REGION Network 163: ACKNOWLEDGE M573-
   RUNG wire#powerrail
      Contact( "M_ZERO" )
      Coil( "DB371_M_UNIT_SPARE".M_CODES_SPARE.Ack_M573 )
   END_RUNG
   // the same network as SCL:
   "DB371_M_UNIT_SPARE".M_CODES_SPARE.Ack_M573 := "M_ZERO";
END_REGION

REGION Network 164: M573-
   RUNG wire#powerrail
      Contact( "DB339_EXTENDED_M_SPARE".M_code[573] )
      wire#w1
      I_Contact( "DB371_M_UNIT_SPARE".M_CODES_SPARE.Ack_M573 )
      I_Contact( "DB2120_MPP_ITC_IPC".RESET_FAULTS )
      I_Contact( "DB371_M_UNIT_SPARE".M_CODES_SPARE.M_RESET_PULSE )
      Coil( "DB371_M_UNIT_SPARE".M_CODES_SPARE.M573 )
   END_RUNG
   RUNG wire#powerrail
      Contact( "DB371_M_UNIT_SPARE".M_CODES_SPARE.M573 )
   END_RUNG wire#w1
   // the same network as SCL:
   "DB371_M_UNIT_SPARE".M_CODES_SPARE.M573 := ("DB339_EXTENDED_M_SPARE".M_code[573] OR "DB371_M_UNIT_SPARE".M_CODES_SPARE.M573) AND NOT "DB371_M_UNIT_SPARE".M_CODES_SPARE.Ack_M573 AND NOT "DB2120_MPP_ITC_IPC".RESET_FAULTS AND NOT "DB371_M_UNIT_SPARE".M_CODES_SPARE.M_RESET_PULSE;
END_REGION

REGION Network 165: ACKNOWLEDGE M574- (READ-IN DISABLE)
   RUNG wire#powerrail
      Contact( "M_ZERO" )
      Coil( "DB371_M_UNIT_SPARE".M_CODES_SPARE.Ack_M574 )
   END_RUNG
   // the same network as SCL:
   "DB371_M_UNIT_SPARE".M_CODES_SPARE.Ack_M574 := "M_ZERO";
END_REGION

REGION Network 166: M574- (READ-IN DISABLE)
   RUNG wire#powerrail
      Contact( "DB339_EXTENDED_M_SPARE".M_code[574] )
      wire#w1
      I_Contact( "DB371_M_UNIT_SPARE".M_CODES_SPARE.Ack_M574 )
      I_Contact( "DB2120_MPP_ITC_IPC".RESET_FAULTS )
      I_Contact( "DB371_M_UNIT_SPARE".M_CODES_SPARE.M_RESET_PULSE )
      Coil( "DB371_M_UNIT_SPARE".M_CODES_SPARE.M574 )
   END_RUNG
   RUNG wire#powerrail
      Contact( "DB371_M_UNIT_SPARE".M_CODES_SPARE.M574 )
   END_RUNG wire#w1
   // the same network as SCL:
   "DB371_M_UNIT_SPARE".M_CODES_SPARE.M574 := ("DB339_EXTENDED_M_SPARE".M_code[574] OR "DB371_M_UNIT_SPARE".M_CODES_SPARE.M574) AND NOT "DB371_M_UNIT_SPARE".M_CODES_SPARE.Ack_M574 AND NOT "DB2120_MPP_ITC_IPC".RESET_FAULTS AND NOT "DB371_M_UNIT_SPARE".M_CODES_SPARE.M_RESET_PULSE;
END_REGION

REGION Network 167: ACKNOWLEDGE M575-(READ-IN DISABLE) / ACKNOWLEDGE M23-SWITCH ON SPINDLE FRAME BLOWING
   RUNG wire#powerrail
      Contact( "M_ZERO" )
      Coil( "DB371_M_UNIT_SPARE".M_CODES_SPARE.Ack_M575 )
   END_RUNG
   // the same network as SCL:
   "DB371_M_UNIT_SPARE".M_CODES_SPARE.Ack_M575 := "M_ZERO";
END_REGION

REGION Network 168: M575-(READ-IN DISABLE) / M23-SWITCH ON SPINDLE FRAME BLOWING
   RUNG wire#powerrail
      Contact( "DB339_EXTENDED_M_SPARE".M_code[575] )
      wire#w1
      I_Contact( "DB371_M_UNIT_SPARE".M_CODES_SPARE.Ack_M575 )
      I_Contact( "DB2120_MPP_ITC_IPC".RESET_FAULTS )
      I_Contact( "DB371_M_UNIT_SPARE".M_CODES_SPARE.M_RESET_PULSE )
      Coil( "DB371_M_UNIT_SPARE".M_CODES_SPARE.M575 )
   END_RUNG
   RUNG wire#powerrail
      Contact( "DB371_M_UNIT_SPARE".M_CODES_SPARE.M575 )
   END_RUNG wire#w1
   // the same network as SCL:
   "DB371_M_UNIT_SPARE".M_CODES_SPARE.M575 := ("DB339_EXTENDED_M_SPARE".M_code[575] OR "DB371_M_UNIT_SPARE".M_CODES_SPARE.M575) AND NOT "DB371_M_UNIT_SPARE".M_CODES_SPARE.Ack_M575 AND NOT "DB2120_MPP_ITC_IPC".RESET_FAULTS AND NOT "DB371_M_UNIT_SPARE".M_CODES_SPARE.M_RESET_PULSE;
END_REGION

REGION Network 169: ACKNOWLEDGE M588- (READ-IN DISABLE) / ACKNOWLEDGE M23-SWITCH ON SPINDLE FRAME BLOWING
   RUNG wire#powerrail
      Contact( "M_ZERO" )
      Coil( "DB371_M_UNIT_SPARE".M_CODES_SPARE.Ack_M588 )
   END_RUNG
   // the same network as SCL:
   "DB371_M_UNIT_SPARE".M_CODES_SPARE.Ack_M588 := "M_ZERO";
END_REGION

REGION Network 170: M588-(READ-IN DISABLE) / M23-SWITCH ON SPINDLE FRAME BLOWING
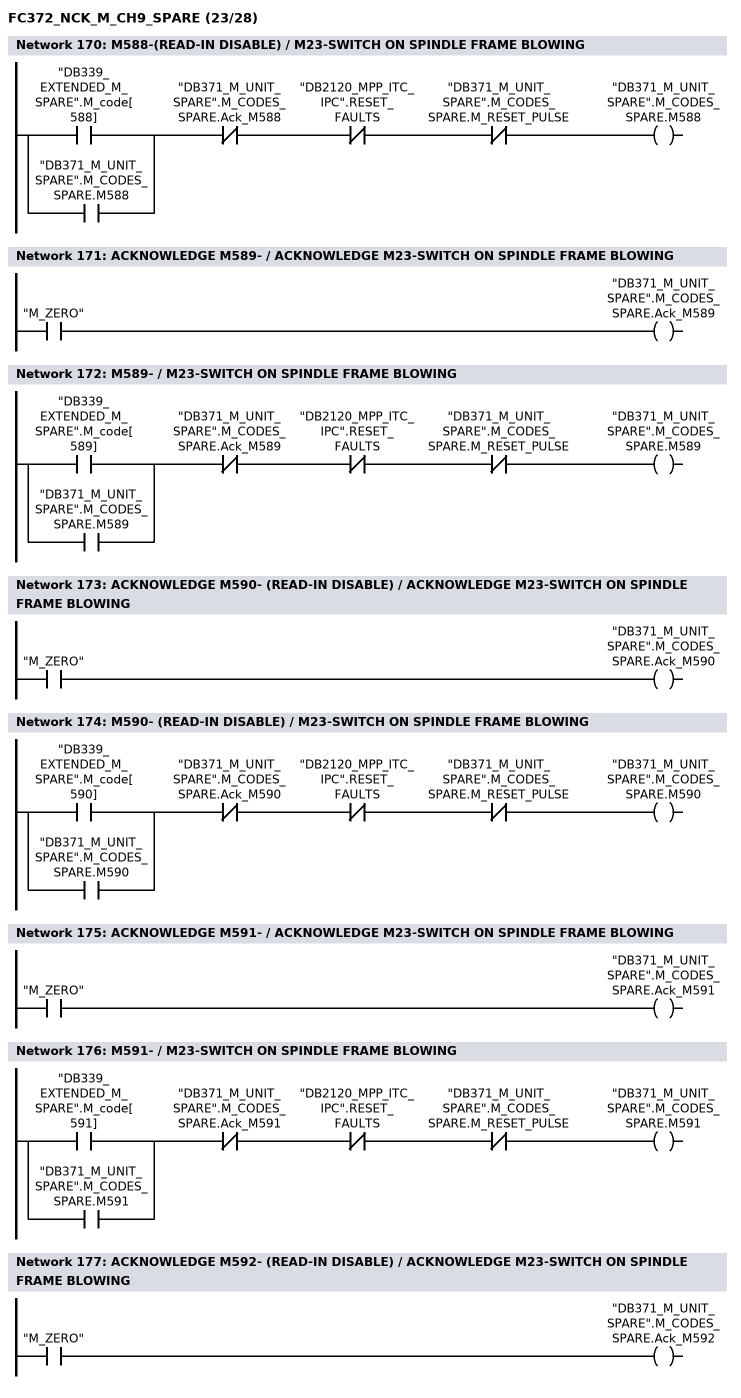
   RUNG wire#powerrail
      Contact( "DB339_EXTENDED_M_SPARE".M_code[588] )
      wire#w1
      I_Contact( "DB371_M_UNIT_SPARE".M_CODES_SPARE.Ack_M588 )
      I_Contact( "DB2120_MPP_ITC_IPC".RESET_FAULTS )
      I_Contact( "DB371_M_UNIT_SPARE".M_CODES_SPARE.M_RESET_PULSE )
      Coil( "DB371_M_UNIT_SPARE".M_CODES_SPARE.M588 )
   END_RUNG
   RUNG wire#powerrail
      Contact( "DB371_M_UNIT_SPARE".M_CODES_SPARE.M588 )
   END_RUNG wire#w1
   // the same network as SCL:
   "DB371_M_UNIT_SPARE".M_CODES_SPARE.M588 := ("DB339_EXTENDED_M_SPARE".M_code[588] OR "DB371_M_UNIT_SPARE".M_CODES_SPARE.M588) AND NOT "DB371_M_UNIT_SPARE".M_CODES_SPARE.Ack_M588 AND NOT "DB2120_MPP_ITC_IPC".RESET_FAULTS AND NOT "DB371_M_UNIT_SPARE".M_CODES_SPARE.M_RESET_PULSE;
END_REGION

REGION Network 171: ACKNOWLEDGE M589- / ACKNOWLEDGE M23-SWITCH ON SPINDLE FRAME BLOWING
   RUNG wire#powerrail
      Contact( "M_ZERO" )
      Coil( "DB371_M_UNIT_SPARE".M_CODES_SPARE.Ack_M589 )
   END_RUNG
   // the same network as SCL:
   "DB371_M_UNIT_SPARE".M_CODES_SPARE.Ack_M589 := "M_ZERO";
END_REGION

REGION Network 172: M589- / M23-SWITCH ON SPINDLE FRAME BLOWING
   RUNG wire#powerrail
      Contact( "DB339_EXTENDED_M_SPARE".M_code[589] )
      wire#w1
      I_Contact( "DB371_M_UNIT_SPARE".M_CODES_SPARE.Ack_M589 )
      I_Contact( "DB2120_MPP_ITC_IPC".RESET_FAULTS )
      I_Contact( "DB371_M_UNIT_SPARE".M_CODES_SPARE.M_RESET_PULSE )
      Coil( "DB371_M_UNIT_SPARE".M_CODES_SPARE.M589 )
   END_RUNG
   RUNG wire#powerrail
      Contact( "DB371_M_UNIT_SPARE".M_CODES_SPARE.M589 )
   END_RUNG wire#w1
   // the same network as SCL:
   "DB371_M_UNIT_SPARE".M_CODES_SPARE.M589 := ("DB339_EXTENDED_M_SPARE".M_code[589] OR "DB371_M_UNIT_SPARE".M_CODES_SPARE.M589) AND NOT "DB371_M_UNIT_SPARE".M_CODES_SPARE.Ack_M589 AND NOT "DB2120_MPP_ITC_IPC".RESET_FAULTS AND NOT "DB371_M_UNIT_SPARE".M_CODES_SPARE.M_RESET_PULSE;
END_REGION

REGION Network 173: ACKNOWLEDGE M590- (READ-IN DISABLE) / ACKNOWLEDGE M23-SWITCH ON SPINDLE FRAME BLOWING
   RUNG wire#powerrail
      Contact( "M_ZERO" )
      Coil( "DB371_M_UNIT_SPARE".M_CODES_SPARE.Ack_M590 )
   END_RUNG
   // the same network as SCL:
   "DB371_M_UNIT_SPARE".M_CODES_SPARE.Ack_M590 := "M_ZERO";
END_REGION

REGION Network 174: M590- (READ-IN DISABLE) / M23-SWITCH ON SPINDLE FRAME BLOWING
   RUNG wire#powerrail
      Contact( "DB339_EXTENDED_M_SPARE".M_code[590] )
      wire#w1
      I_Contact( "DB371_M_UNIT_SPARE".M_CODES_SPARE.Ack_M590 )
      I_Contact( "DB2120_MPP_ITC_IPC".RESET_FAULTS )
      I_Contact( "DB371_M_UNIT_SPARE".M_CODES_SPARE.M_RESET_PULSE )
      Coil( "DB371_M_UNIT_SPARE".M_CODES_SPARE.M590 )
   END_RUNG
   RUNG wire#powerrail
      Contact( "DB371_M_UNIT_SPARE".M_CODES_SPARE.M590 )
   END_RUNG wire#w1
   // the same network as SCL:
   "DB371_M_UNIT_SPARE".M_CODES_SPARE.M590 := ("DB339_EXTENDED_M_SPARE".M_code[590] OR "DB371_M_UNIT_SPARE".M_CODES_SPARE.M590) AND NOT "DB371_M_UNIT_SPARE".M_CODES_SPARE.Ack_M590 AND NOT "DB2120_MPP_ITC_IPC".RESET_FAULTS AND NOT "DB371_M_UNIT_SPARE".M_CODES_SPARE.M_RESET_PULSE;
END_REGION

REGION Network 175: ACKNOWLEDGE M591- / ACKNOWLEDGE M23-SWITCH ON SPINDLE FRAME BLOWING
   RUNG wire#powerrail
      Contact( "M_ZERO" )
      Coil( "DB371_M_UNIT_SPARE".M_CODES_SPARE.Ack_M591 )
   END_RUNG
   // the same network as SCL:
   "DB371_M_UNIT_SPARE".M_CODES_SPARE.Ack_M591 := "M_ZERO";
END_REGION

REGION Network 176: M591- / M23-SWITCH ON SPINDLE FRAME BLOWING
   RUNG wire#powerrail
      Contact( "DB339_EXTENDED_M_SPARE".M_code[591] )
      wire#w1
      I_Contact( "DB371_M_UNIT_SPARE".M_CODES_SPARE.Ack_M591 )
      I_Contact( "DB2120_MPP_ITC_IPC".RESET_FAULTS )
      I_Contact( "DB371_M_UNIT_SPARE".M_CODES_SPARE.M_RESET_PULSE )
      Coil( "DB371_M_UNIT_SPARE".M_CODES_SPARE.M591 )
   END_RUNG
   RUNG wire#powerrail
      Contact( "DB371_M_UNIT_SPARE".M_CODES_SPARE.M591 )
   END_RUNG wire#w1
   // the same network as SCL:
   "DB371_M_UNIT_SPARE".M_CODES_SPARE.M591 := ("DB339_EXTENDED_M_SPARE".M_code[591] OR "DB371_M_UNIT_SPARE".M_CODES_SPARE.M591) AND NOT "DB371_M_UNIT_SPARE".M_CODES_SPARE.Ack_M591 AND NOT "DB2120_MPP_ITC_IPC".RESET_FAULTS AND NOT "DB371_M_UNIT_SPARE".M_CODES_SPARE.M_RESET_PULSE;
END_REGION

REGION Network 177: ACKNOWLEDGE M592- (READ-IN DISABLE) / ACKNOWLEDGE M23-SWITCH ON SPINDLE FRAME BLOWING
   RUNG wire#powerrail
      Contact( "M_ZERO" )
      Coil( "DB371_M_UNIT_SPARE".M_CODES_SPARE.Ack_M592 )
   END_RUNG
   // the same network as SCL:
   "DB371_M_UNIT_SPARE".M_CODES_SPARE.Ack_M592 := "M_ZERO";
END_REGION

REGION Network 178: M592- (READ-IN DISABLE) / M23-SWITCH ON SPINDLE FRAME BLOWING
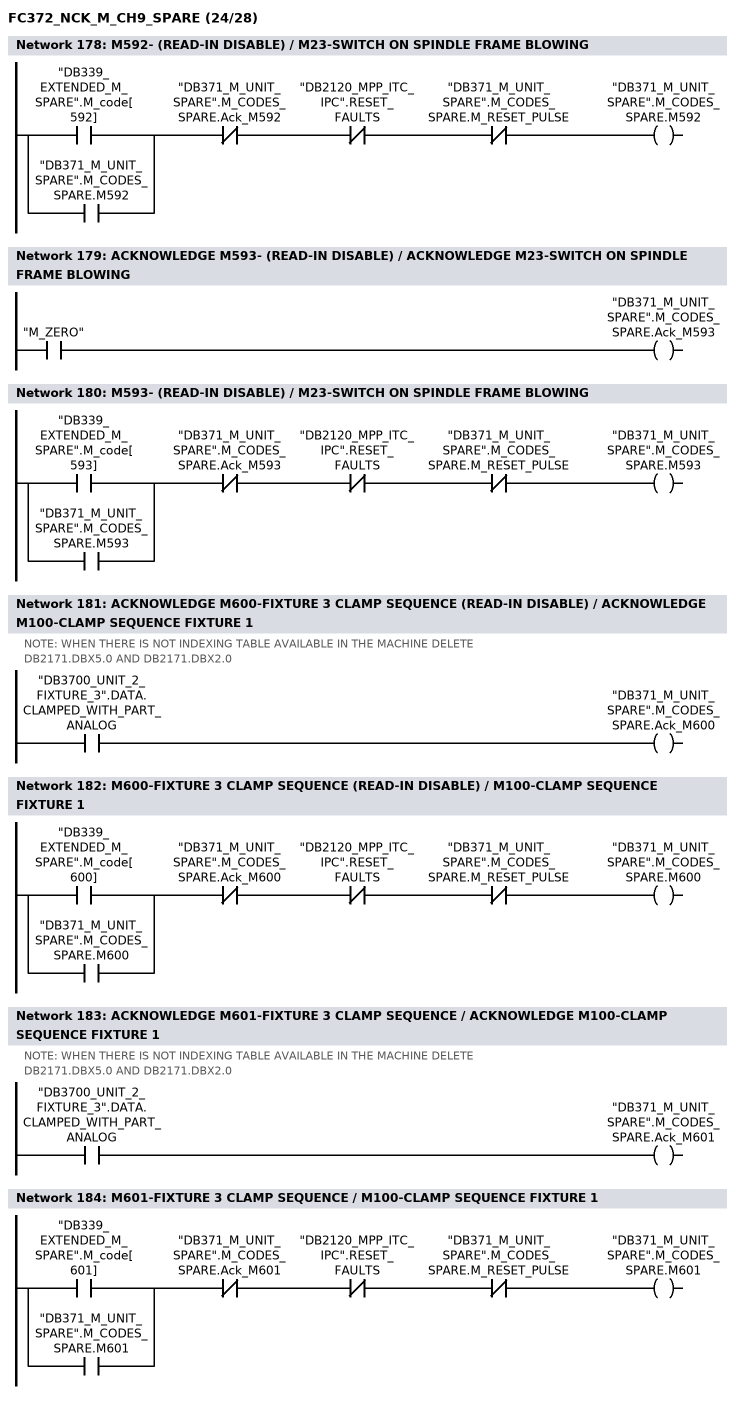
   RUNG wire#powerrail
      Contact( "DB339_EXTENDED_M_SPARE".M_code[592] )
      wire#w1
      I_Contact( "DB371_M_UNIT_SPARE".M_CODES_SPARE.Ack_M592 )
      I_Contact( "DB2120_MPP_ITC_IPC".RESET_FAULTS )
      I_Contact( "DB371_M_UNIT_SPARE".M_CODES_SPARE.M_RESET_PULSE )
      Coil( "DB371_M_UNIT_SPARE".M_CODES_SPARE.M592 )
   END_RUNG
   RUNG wire#powerrail
      Contact( "DB371_M_UNIT_SPARE".M_CODES_SPARE.M592 )
   END_RUNG wire#w1
   // the same network as SCL:
   "DB371_M_UNIT_SPARE".M_CODES_SPARE.M592 := ("DB339_EXTENDED_M_SPARE".M_code[592] OR "DB371_M_UNIT_SPARE".M_CODES_SPARE.M592) AND NOT "DB371_M_UNIT_SPARE".M_CODES_SPARE.Ack_M592 AND NOT "DB2120_MPP_ITC_IPC".RESET_FAULTS AND NOT "DB371_M_UNIT_SPARE".M_CODES_SPARE.M_RESET_PULSE;
END_REGION

REGION Network 179: ACKNOWLEDGE M593- (READ-IN DISABLE) / ACKNOWLEDGE M23-SWITCH ON SPINDLE FRAME BLOWING
   RUNG wire#powerrail
      Contact( "M_ZERO" )
      Coil( "DB371_M_UNIT_SPARE".M_CODES_SPARE.Ack_M593 )
   END_RUNG
   // the same network as SCL:
   "DB371_M_UNIT_SPARE".M_CODES_SPARE.Ack_M593 := "M_ZERO";
END_REGION

REGION Network 180: M593- (READ-IN DISABLE) / M23-SWITCH ON SPINDLE FRAME BLOWING
   RUNG wire#powerrail
      Contact( "DB339_EXTENDED_M_SPARE".M_code[593] )
      wire#w1
      I_Contact( "DB371_M_UNIT_SPARE".M_CODES_SPARE.Ack_M593 )
      I_Contact( "DB2120_MPP_ITC_IPC".RESET_FAULTS )
      I_Contact( "DB371_M_UNIT_SPARE".M_CODES_SPARE.M_RESET_PULSE )
      Coil( "DB371_M_UNIT_SPARE".M_CODES_SPARE.M593 )
   END_RUNG
   RUNG wire#powerrail
      Contact( "DB371_M_UNIT_SPARE".M_CODES_SPARE.M593 )
   END_RUNG wire#w1
   // the same network as SCL:
   "DB371_M_UNIT_SPARE".M_CODES_SPARE.M593 := ("DB339_EXTENDED_M_SPARE".M_code[593] OR "DB371_M_UNIT_SPARE".M_CODES_SPARE.M593) AND NOT "DB371_M_UNIT_SPARE".M_CODES_SPARE.Ack_M593 AND NOT "DB2120_MPP_ITC_IPC".RESET_FAULTS AND NOT "DB371_M_UNIT_SPARE".M_CODES_SPARE.M_RESET_PULSE;
END_REGION

REGION Network 181: ACKNOWLEDGE M600-FIXTURE 3 CLAMP SEQUENCE (READ-IN DISABLE) / ACKNOWLEDGE M100-CLAMP SEQUENCE FIXTURE 1
   // NOTE: WHEN THERE IS NOT INDEXING TABLE AVAILABLE IN THE MACHINE DELETE 
   // DB2171.DBX5.0 AND DB2171.DBX2.0
   RUNG wire#powerrail
      Contact( "DB3700_UNIT_2_FIXTURE_3".DATA.CLAMPED_WITH_PART_ANALOG )
      Coil( "DB371_M_UNIT_SPARE".M_CODES_SPARE.Ack_M600 )
   END_RUNG
   // the same network as SCL:
   "DB371_M_UNIT_SPARE".M_CODES_SPARE.Ack_M600 := "DB3700_UNIT_2_FIXTURE_3".DATA.CLAMPED_WITH_PART_ANALOG;
END_REGION

REGION Network 182: M600-FIXTURE 3 CLAMP SEQUENCE (READ-IN DISABLE) / M100-CLAMP SEQUENCE FIXTURE 1
   RUNG wire#powerrail
      Contact( "DB339_EXTENDED_M_SPARE".M_code[600] )
      wire#w1
      I_Contact( "DB371_M_UNIT_SPARE".M_CODES_SPARE.Ack_M600 )
      I_Contact( "DB2120_MPP_ITC_IPC".RESET_FAULTS )
      I_Contact( "DB371_M_UNIT_SPARE".M_CODES_SPARE.M_RESET_PULSE )
      Coil( "DB371_M_UNIT_SPARE".M_CODES_SPARE.M600 )
   END_RUNG
   RUNG wire#powerrail
      Contact( "DB371_M_UNIT_SPARE".M_CODES_SPARE.M600 )
   END_RUNG wire#w1
   // the same network as SCL:
   "DB371_M_UNIT_SPARE".M_CODES_SPARE.M600 := ("DB339_EXTENDED_M_SPARE".M_code[600] OR "DB371_M_UNIT_SPARE".M_CODES_SPARE.M600) AND NOT "DB371_M_UNIT_SPARE".M_CODES_SPARE.Ack_M600 AND NOT "DB2120_MPP_ITC_IPC".RESET_FAULTS AND NOT "DB371_M_UNIT_SPARE".M_CODES_SPARE.M_RESET_PULSE;
END_REGION

REGION Network 183: ACKNOWLEDGE M601-FIXTURE 3 CLAMP SEQUENCE / ACKNOWLEDGE M100-CLAMP SEQUENCE FIXTURE 1
   // NOTE: WHEN THERE IS NOT INDEXING TABLE AVAILABLE IN THE MACHINE DELETE 
   // DB2171.DBX5.0 AND DB2171.DBX2.0
   RUNG wire#powerrail
      Contact( "DB3700_UNIT_2_FIXTURE_3".DATA.CLAMPED_WITH_PART_ANALOG )
      Coil( "DB371_M_UNIT_SPARE".M_CODES_SPARE.Ack_M601 )
   END_RUNG
   // the same network as SCL:
   "DB371_M_UNIT_SPARE".M_CODES_SPARE.Ack_M601 := "DB3700_UNIT_2_FIXTURE_3".DATA.CLAMPED_WITH_PART_ANALOG;
END_REGION

REGION Network 184: M601-FIXTURE 3 CLAMP SEQUENCE / M100-CLAMP SEQUENCE FIXTURE 1
   RUNG wire#powerrail
      Contact( "DB339_EXTENDED_M_SPARE".M_code[601] )
      wire#w1
      I_Contact( "DB371_M_UNIT_SPARE".M_CODES_SPARE.Ack_M601 )
      I_Contact( "DB2120_MPP_ITC_IPC".RESET_FAULTS )
      I_Contact( "DB371_M_UNIT_SPARE".M_CODES_SPARE.M_RESET_PULSE )
      Coil( "DB371_M_UNIT_SPARE".M_CODES_SPARE.M601 )
   END_RUNG
   RUNG wire#powerrail
      Contact( "DB371_M_UNIT_SPARE".M_CODES_SPARE.M601 )
   END_RUNG wire#w1
   // the same network as SCL:
   "DB371_M_UNIT_SPARE".M_CODES_SPARE.M601 := ("DB339_EXTENDED_M_SPARE".M_code[601] OR "DB371_M_UNIT_SPARE".M_CODES_SPARE.M601) AND NOT "DB371_M_UNIT_SPARE".M_CODES_SPARE.Ack_M601 AND NOT "DB2120_MPP_ITC_IPC".RESET_FAULTS AND NOT "DB371_M_UNIT_SPARE".M_CODES_SPARE.M_RESET_PULSE;
END_REGION

REGION Network 185: ACKNOWLEDGE M602-FIXTURE 3 UNCLAMP SEQUENCE (READ-IN DISABLE) / ACKNOWLEDGE M101-UNCLAMP SEQUENCE FIXTURE 1
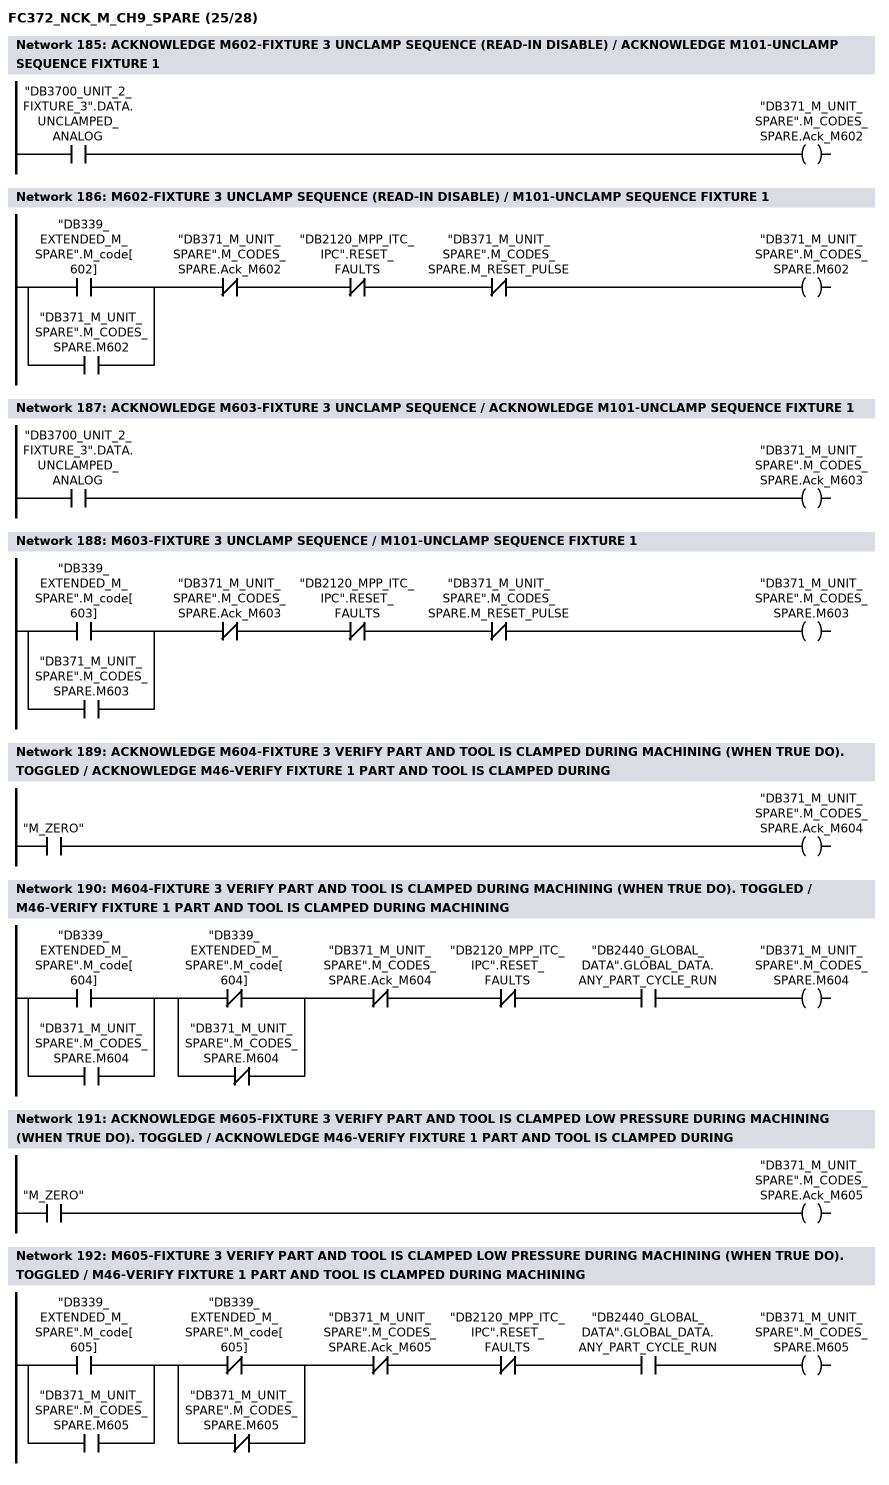
   RUNG wire#powerrail
      Contact( "DB3700_UNIT_2_FIXTURE_3".DATA.UNCLAMPED_ANALOG )
      Coil( "DB371_M_UNIT_SPARE".M_CODES_SPARE.Ack_M602 )
   END_RUNG
   // the same network as SCL:
   "DB371_M_UNIT_SPARE".M_CODES_SPARE.Ack_M602 := "DB3700_UNIT_2_FIXTURE_3".DATA.UNCLAMPED_ANALOG;
END_REGION

REGION Network 186: M602-FIXTURE 3 UNCLAMP SEQUENCE (READ-IN DISABLE) / M101-UNCLAMP SEQUENCE FIXTURE 1
   RUNG wire#powerrail
      Contact( "DB339_EXTENDED_M_SPARE".M_code[602] )
      wire#w1
      I_Contact( "DB371_M_UNIT_SPARE".M_CODES_SPARE.Ack_M602 )
      I_Contact( "DB2120_MPP_ITC_IPC".RESET_FAULTS )
      I_Contact( "DB371_M_UNIT_SPARE".M_CODES_SPARE.M_RESET_PULSE )
      Coil( "DB371_M_UNIT_SPARE".M_CODES_SPARE.M602 )
   END_RUNG
   RUNG wire#powerrail
      Contact( "DB371_M_UNIT_SPARE".M_CODES_SPARE.M602 )
   END_RUNG wire#w1
   // the same network as SCL:
   "DB371_M_UNIT_SPARE".M_CODES_SPARE.M602 := ("DB339_EXTENDED_M_SPARE".M_code[602] OR "DB371_M_UNIT_SPARE".M_CODES_SPARE.M602) AND NOT "DB371_M_UNIT_SPARE".M_CODES_SPARE.Ack_M602 AND NOT "DB2120_MPP_ITC_IPC".RESET_FAULTS AND NOT "DB371_M_UNIT_SPARE".M_CODES_SPARE.M_RESET_PULSE;
END_REGION

REGION Network 187: ACKNOWLEDGE M603-FIXTURE 3 UNCLAMP SEQUENCE / ACKNOWLEDGE M101-UNCLAMP SEQUENCE FIXTURE 1
   RUNG wire#powerrail
      Contact( "DB3700_UNIT_2_FIXTURE_3".DATA.UNCLAMPED_ANALOG )
      Coil( "DB371_M_UNIT_SPARE".M_CODES_SPARE.Ack_M603 )
   END_RUNG
   // the same network as SCL:
   "DB371_M_UNIT_SPARE".M_CODES_SPARE.Ack_M603 := "DB3700_UNIT_2_FIXTURE_3".DATA.UNCLAMPED_ANALOG;
END_REGION

REGION Network 188: M603-FIXTURE 3 UNCLAMP SEQUENCE / M101-UNCLAMP SEQUENCE FIXTURE 1
   RUNG wire#powerrail
      Contact( "DB339_EXTENDED_M_SPARE".M_code[603] )
      wire#w1
      I_Contact( "DB371_M_UNIT_SPARE".M_CODES_SPARE.Ack_M603 )
      I_Contact( "DB2120_MPP_ITC_IPC".RESET_FAULTS )
      I_Contact( "DB371_M_UNIT_SPARE".M_CODES_SPARE.M_RESET_PULSE )
      Coil( "DB371_M_UNIT_SPARE".M_CODES_SPARE.M603 )
   END_RUNG
   RUNG wire#powerrail
      Contact( "DB371_M_UNIT_SPARE".M_CODES_SPARE.M603 )
   END_RUNG wire#w1
   // the same network as SCL:
   "DB371_M_UNIT_SPARE".M_CODES_SPARE.M603 := ("DB339_EXTENDED_M_SPARE".M_code[603] OR "DB371_M_UNIT_SPARE".M_CODES_SPARE.M603) AND NOT "DB371_M_UNIT_SPARE".M_CODES_SPARE.Ack_M603 AND NOT "DB2120_MPP_ITC_IPC".RESET_FAULTS AND NOT "DB371_M_UNIT_SPARE".M_CODES_SPARE.M_RESET_PULSE;
END_REGION

REGION Network 189: ACKNOWLEDGE M604-FIXTURE 3 VERIFY PART AND TOOL IS CLAMPED DURING MACHINING (WHEN TRUE DO). TOGGLED / ACKNOWLEDGE M46-VERIFY FIXTURE 1 PART AND TOOL IS CLAMPED DURING
   RUNG wire#powerrail
      Contact( "M_ZERO" )
      Coil( "DB371_M_UNIT_SPARE".M_CODES_SPARE.Ack_M604 )
   END_RUNG
   // the same network as SCL:
   "DB371_M_UNIT_SPARE".M_CODES_SPARE.Ack_M604 := "M_ZERO";
END_REGION

REGION Network 190: M604-FIXTURE 3 VERIFY PART AND TOOL IS CLAMPED DURING MACHINING (WHEN TRUE DO). TOGGLED / M46-VERIFY FIXTURE 1 PART AND TOOL IS CLAMPED DURING MACHINING
   RUNG wire#powerrail
      Contact( "DB339_EXTENDED_M_SPARE".M_code[604] )
      wire#w1
      I_Contact( "DB339_EXTENDED_M_SPARE".M_code[604] )
      wire#w2
      I_Contact( "DB371_M_UNIT_SPARE".M_CODES_SPARE.Ack_M604 )
      I_Contact( "DB2120_MPP_ITC_IPC".RESET_FAULTS )
      Contact( "DB2440_GLOBAL_DATA".GLOBAL_DATA.ANY_PART_CYCLE_RUN )
      Coil( "DB371_M_UNIT_SPARE".M_CODES_SPARE.M604 )
   END_RUNG
   RUNG wire#powerrail
      Contact( "DB371_M_UNIT_SPARE".M_CODES_SPARE.M604 )
   END_RUNG wire#w1
   RUNG wire#w1
      I_Contact( "DB371_M_UNIT_SPARE".M_CODES_SPARE.M604 )
   END_RUNG wire#w2
   // the same network as SCL:
   "DB371_M_UNIT_SPARE".M_CODES_SPARE.M604 := ("DB339_EXTENDED_M_SPARE".M_code[604] OR "DB371_M_UNIT_SPARE".M_CODES_SPARE.M604) AND (NOT "DB339_EXTENDED_M_SPARE".M_code[604] OR NOT "DB371_M_UNIT_SPARE".M_CODES_SPARE.M604) AND NOT "DB371_M_UNIT_SPARE".M_CODES_SPARE.Ack_M604 AND NOT "DB2120_MPP_ITC_IPC".RESET_FAULTS AND "DB2440_GLOBAL_DATA".GLOBAL_DATA.ANY_PART_CYCLE_RUN;
END_REGION

REGION Network 191: ACKNOWLEDGE M605-FIXTURE 3 VERIFY PART AND TOOL IS CLAMPED LOW PRESSURE DURING MACHINING (WHEN TRUE DO). TOGGLED / ACKNOWLEDGE M46-VERIFY FIXTURE 1 PART AND TOOL IS CLAMPED DURING
   RUNG wire#powerrail
      Contact( "M_ZERO" )
      Coil( "DB371_M_UNIT_SPARE".M_CODES_SPARE.Ack_M605 )
   END_RUNG
   // the same network as SCL:
   "DB371_M_UNIT_SPARE".M_CODES_SPARE.Ack_M605 := "M_ZERO";
END_REGION

REGION Network 192: M605-FIXTURE 3 VERIFY PART AND TOOL IS CLAMPED LOW PRESSURE DURING MACHINING (WHEN TRUE DO). TOGGLED / M46-VERIFY FIXTURE 1 PART AND TOOL IS CLAMPED DURING MACHINING
   RUNG wire#powerrail
      Contact( "DB339_EXTENDED_M_SPARE".M_code[605] )
      wire#w1
      I_Contact( "DB339_EXTENDED_M_SPARE".M_code[605] )
      wire#w2
      I_Contact( "DB371_M_UNIT_SPARE".M_CODES_SPARE.Ack_M605 )
      I_Contact( "DB2120_MPP_ITC_IPC".RESET_FAULTS )
      Contact( "DB2440_GLOBAL_DATA".GLOBAL_DATA.ANY_PART_CYCLE_RUN )
      Coil( "DB371_M_UNIT_SPARE".M_CODES_SPARE.M605 )
   END_RUNG
   RUNG wire#powerrail
      Contact( "DB371_M_UNIT_SPARE".M_CODES_SPARE.M605 )
   END_RUNG wire#w1
   RUNG wire#w1
      I_Contact( "DB371_M_UNIT_SPARE".M_CODES_SPARE.M605 )
   END_RUNG wire#w2
   // the same network as SCL:
   "DB371_M_UNIT_SPARE".M_CODES_SPARE.M605 := ("DB339_EXTENDED_M_SPARE".M_code[605] OR "DB371_M_UNIT_SPARE".M_CODES_SPARE.M605) AND (NOT "DB339_EXTENDED_M_SPARE".M_code[605] OR NOT "DB371_M_UNIT_SPARE".M_CODES_SPARE.M605) AND NOT "DB371_M_UNIT_SPARE".M_CODES_SPARE.Ack_M605 AND NOT "DB2120_MPP_ITC_IPC".RESET_FAULTS AND "DB2440_GLOBAL_DATA".GLOBAL_DATA.ANY_PART_CYCLE_RUN;
END_REGION

REGION Network 193: ACKNOWLEDGE M606-FIXTURE 3 VERIFY PARTS ARE UNCLAMPED PARTS LOADING (WHEN TRUE DO). TOGGLED / ACKNOWLEDGE M47-VERIFY FIXTURE 2 PART AND TOOL IS CLAMPED DURING
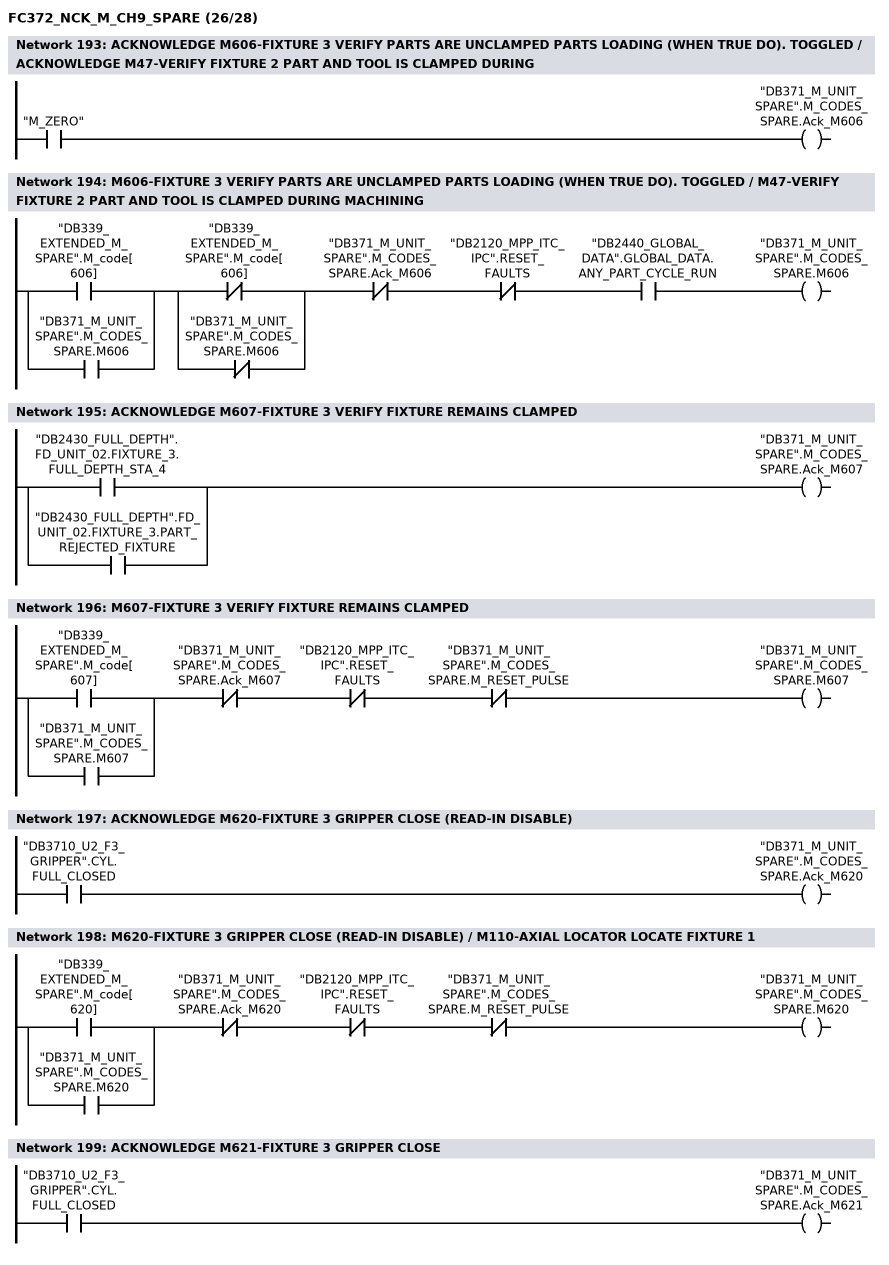
   RUNG wire#powerrail
      Contact( "M_ZERO" )
      Coil( "DB371_M_UNIT_SPARE".M_CODES_SPARE.Ack_M606 )
   END_RUNG
   // the same network as SCL:
   "DB371_M_UNIT_SPARE".M_CODES_SPARE.Ack_M606 := "M_ZERO";
END_REGION

REGION Network 194: M606-FIXTURE 3 VERIFY PARTS ARE UNCLAMPED PARTS LOADING (WHEN TRUE DO). TOGGLED / M47-VERIFY FIXTURE 2 PART AND TOOL IS CLAMPED DURING MACHINING
   RUNG wire#powerrail
      Contact( "DB339_EXTENDED_M_SPARE".M_code[606] )
      wire#w1
      I_Contact( "DB339_EXTENDED_M_SPARE".M_code[606] )
      wire#w2
      I_Contact( "DB371_M_UNIT_SPARE".M_CODES_SPARE.Ack_M606 )
      I_Contact( "DB2120_MPP_ITC_IPC".RESET_FAULTS )
      Contact( "DB2440_GLOBAL_DATA".GLOBAL_DATA.ANY_PART_CYCLE_RUN )
      Coil( "DB371_M_UNIT_SPARE".M_CODES_SPARE.M606 )
   END_RUNG
   RUNG wire#powerrail
      Contact( "DB371_M_UNIT_SPARE".M_CODES_SPARE.M606 )
   END_RUNG wire#w1
   RUNG wire#w1
      I_Contact( "DB371_M_UNIT_SPARE".M_CODES_SPARE.M606 )
   END_RUNG wire#w2
   // the same network as SCL:
   "DB371_M_UNIT_SPARE".M_CODES_SPARE.M606 := ("DB339_EXTENDED_M_SPARE".M_code[606] OR "DB371_M_UNIT_SPARE".M_CODES_SPARE.M606) AND (NOT "DB339_EXTENDED_M_SPARE".M_code[606] OR NOT "DB371_M_UNIT_SPARE".M_CODES_SPARE.M606) AND NOT "DB371_M_UNIT_SPARE".M_CODES_SPARE.Ack_M606 AND NOT "DB2120_MPP_ITC_IPC".RESET_FAULTS AND "DB2440_GLOBAL_DATA".GLOBAL_DATA.ANY_PART_CYCLE_RUN;
END_REGION

REGION Network 195: ACKNOWLEDGE M607-FIXTURE 3 VERIFY FIXTURE REMAINS CLAMPED
   RUNG wire#powerrail
      Contact( "DB2430_FULL_DEPTH".FD_UNIT_02.FIXTURE_3.FULL_DEPTH_STA_4 )
      wire#w1
      Coil( "DB371_M_UNIT_SPARE".M_CODES_SPARE.Ack_M607 )
   END_RUNG
   RUNG wire#powerrail
      Contact( "DB2430_FULL_DEPTH".FD_UNIT_02.FIXTURE_3.PART_REJECTED_FIXTURE )
   END_RUNG wire#w1
   // the same network as SCL:
   "DB371_M_UNIT_SPARE".M_CODES_SPARE.Ack_M607 := "DB2430_FULL_DEPTH".FD_UNIT_02.FIXTURE_3.FULL_DEPTH_STA_4 OR "DB2430_FULL_DEPTH".FD_UNIT_02.FIXTURE_3.PART_REJECTED_FIXTURE;
END_REGION

REGION Network 196: M607-FIXTURE 3 VERIFY FIXTURE REMAINS CLAMPED
   RUNG wire#powerrail
      Contact( "DB339_EXTENDED_M_SPARE".M_code[607] )
      wire#w1
      I_Contact( "DB371_M_UNIT_SPARE".M_CODES_SPARE.Ack_M607 )
      I_Contact( "DB2120_MPP_ITC_IPC".RESET_FAULTS )
      I_Contact( "DB371_M_UNIT_SPARE".M_CODES_SPARE.M_RESET_PULSE )
      Coil( "DB371_M_UNIT_SPARE".M_CODES_SPARE.M607 )
   END_RUNG
   RUNG wire#powerrail
      Contact( "DB371_M_UNIT_SPARE".M_CODES_SPARE.M607 )
   END_RUNG wire#w1
   // the same network as SCL:
   "DB371_M_UNIT_SPARE".M_CODES_SPARE.M607 := ("DB339_EXTENDED_M_SPARE".M_code[607] OR "DB371_M_UNIT_SPARE".M_CODES_SPARE.M607) AND NOT "DB371_M_UNIT_SPARE".M_CODES_SPARE.Ack_M607 AND NOT "DB2120_MPP_ITC_IPC".RESET_FAULTS AND NOT "DB371_M_UNIT_SPARE".M_CODES_SPARE.M_RESET_PULSE;
END_REGION

REGION Network 197: ACKNOWLEDGE M620-FIXTURE 3 GRIPPER CLOSE (READ-IN DISABLE)
   RUNG wire#powerrail
      Contact( "DB3710_U2_F3_GRIPPER".CYL.FULL_CLOSED )
      Coil( "DB371_M_UNIT_SPARE".M_CODES_SPARE.Ack_M620 )
   END_RUNG
   // the same network as SCL:
   "DB371_M_UNIT_SPARE".M_CODES_SPARE.Ack_M620 := "DB3710_U2_F3_GRIPPER".CYL.FULL_CLOSED;
END_REGION

REGION Network 198: M620-FIXTURE 3 GRIPPER CLOSE (READ-IN DISABLE) / M110-AXIAL LOCATOR LOCATE FIXTURE 1
   RUNG wire#powerrail
      Contact( "DB339_EXTENDED_M_SPARE".M_code[620] )
      wire#w1
      I_Contact( "DB371_M_UNIT_SPARE".M_CODES_SPARE.Ack_M620 )
      I_Contact( "DB2120_MPP_ITC_IPC".RESET_FAULTS )
      I_Contact( "DB371_M_UNIT_SPARE".M_CODES_SPARE.M_RESET_PULSE )
      Coil( "DB371_M_UNIT_SPARE".M_CODES_SPARE.M620 )
   END_RUNG
   RUNG wire#powerrail
      Contact( "DB371_M_UNIT_SPARE".M_CODES_SPARE.M620 )
   END_RUNG wire#w1
   // the same network as SCL:
   "DB371_M_UNIT_SPARE".M_CODES_SPARE.M620 := ("DB339_EXTENDED_M_SPARE".M_code[620] OR "DB371_M_UNIT_SPARE".M_CODES_SPARE.M620) AND NOT "DB371_M_UNIT_SPARE".M_CODES_SPARE.Ack_M620 AND NOT "DB2120_MPP_ITC_IPC".RESET_FAULTS AND NOT "DB371_M_UNIT_SPARE".M_CODES_SPARE.M_RESET_PULSE;
END_REGION

REGION Network 199: ACKNOWLEDGE M621-FIXTURE 3 GRIPPER CLOSE
   RUNG wire#powerrail
      Contact( "DB3710_U2_F3_GRIPPER".CYL.FULL_CLOSED )
      Coil( "DB371_M_UNIT_SPARE".M_CODES_SPARE.Ack_M621 )
   END_RUNG
   // the same network as SCL:
   "DB371_M_UNIT_SPARE".M_CODES_SPARE.Ack_M621 := "DB3710_U2_F3_GRIPPER".CYL.FULL_CLOSED;
END_REGION

REGION Network 200: M621-FIXTURE 3 GRIPPER CLOSE / M110-AXIAL LOCATOR LOCATE FIXTURE 1
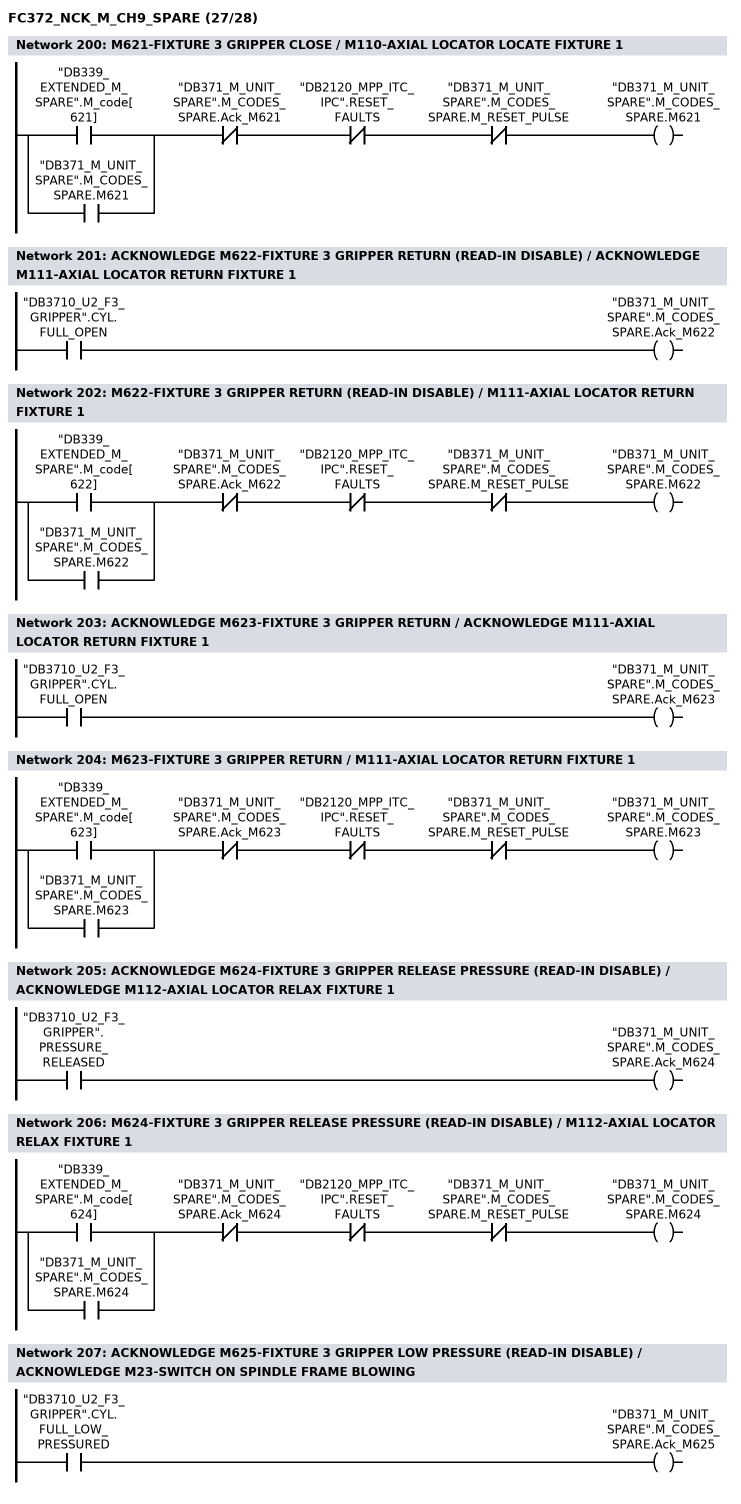
   RUNG wire#powerrail
      Contact( "DB339_EXTENDED_M_SPARE".M_code[621] )
      wire#w1
      I_Contact( "DB371_M_UNIT_SPARE".M_CODES_SPARE.Ack_M621 )
      I_Contact( "DB2120_MPP_ITC_IPC".RESET_FAULTS )
      I_Contact( "DB371_M_UNIT_SPARE".M_CODES_SPARE.M_RESET_PULSE )
      Coil( "DB371_M_UNIT_SPARE".M_CODES_SPARE.M621 )
   END_RUNG
   RUNG wire#powerrail
      Contact( "DB371_M_UNIT_SPARE".M_CODES_SPARE.M621 )
   END_RUNG wire#w1
   // the same network as SCL:
   "DB371_M_UNIT_SPARE".M_CODES_SPARE.M621 := ("DB339_EXTENDED_M_SPARE".M_code[621] OR "DB371_M_UNIT_SPARE".M_CODES_SPARE.M621) AND NOT "DB371_M_UNIT_SPARE".M_CODES_SPARE.Ack_M621 AND NOT "DB2120_MPP_ITC_IPC".RESET_FAULTS AND NOT "DB371_M_UNIT_SPARE".M_CODES_SPARE.M_RESET_PULSE;
END_REGION

REGION Network 201: ACKNOWLEDGE M622-FIXTURE 3 GRIPPER RETURN (READ-IN DISABLE) / ACKNOWLEDGE M111-AXIAL LOCATOR RETURN FIXTURE 1
   RUNG wire#powerrail
      Contact( "DB3710_U2_F3_GRIPPER".CYL.FULL_OPEN )
      Coil( "DB371_M_UNIT_SPARE".M_CODES_SPARE.Ack_M622 )
   END_RUNG
   // the same network as SCL:
   "DB371_M_UNIT_SPARE".M_CODES_SPARE.Ack_M622 := "DB3710_U2_F3_GRIPPER".CYL.FULL_OPEN;
END_REGION

REGION Network 202: M622-FIXTURE 3 GRIPPER RETURN (READ-IN DISABLE) / M111-AXIAL LOCATOR RETURN FIXTURE 1
   RUNG wire#powerrail
      Contact( "DB339_EXTENDED_M_SPARE".M_code[622] )
      wire#w1
      I_Contact( "DB371_M_UNIT_SPARE".M_CODES_SPARE.Ack_M622 )
      I_Contact( "DB2120_MPP_ITC_IPC".RESET_FAULTS )
      I_Contact( "DB371_M_UNIT_SPARE".M_CODES_SPARE.M_RESET_PULSE )
      Coil( "DB371_M_UNIT_SPARE".M_CODES_SPARE.M622 )
   END_RUNG
   RUNG wire#powerrail
      Contact( "DB371_M_UNIT_SPARE".M_CODES_SPARE.M622 )
   END_RUNG wire#w1
   // the same network as SCL:
   "DB371_M_UNIT_SPARE".M_CODES_SPARE.M622 := ("DB339_EXTENDED_M_SPARE".M_code[622] OR "DB371_M_UNIT_SPARE".M_CODES_SPARE.M622) AND NOT "DB371_M_UNIT_SPARE".M_CODES_SPARE.Ack_M622 AND NOT "DB2120_MPP_ITC_IPC".RESET_FAULTS AND NOT "DB371_M_UNIT_SPARE".M_CODES_SPARE.M_RESET_PULSE;
END_REGION

REGION Network 203: ACKNOWLEDGE M623-FIXTURE 3 GRIPPER RETURN / ACKNOWLEDGE M111-AXIAL LOCATOR RETURN FIXTURE 1
   RUNG wire#powerrail
      Contact( "DB3710_U2_F3_GRIPPER".CYL.FULL_OPEN )
      Coil( "DB371_M_UNIT_SPARE".M_CODES_SPARE.Ack_M623 )
   END_RUNG
   // the same network as SCL:
   "DB371_M_UNIT_SPARE".M_CODES_SPARE.Ack_M623 := "DB3710_U2_F3_GRIPPER".CYL.FULL_OPEN;
END_REGION

REGION Network 204: M623-FIXTURE 3 GRIPPER RETURN / M111-AXIAL LOCATOR RETURN FIXTURE 1
   RUNG wire#powerrail
      Contact( "DB339_EXTENDED_M_SPARE".M_code[623] )
      wire#w1
      I_Contact( "DB371_M_UNIT_SPARE".M_CODES_SPARE.Ack_M623 )
      I_Contact( "DB2120_MPP_ITC_IPC".RESET_FAULTS )
      I_Contact( "DB371_M_UNIT_SPARE".M_CODES_SPARE.M_RESET_PULSE )
      Coil( "DB371_M_UNIT_SPARE".M_CODES_SPARE.M623 )
   END_RUNG
   RUNG wire#powerrail
      Contact( "DB371_M_UNIT_SPARE".M_CODES_SPARE.M623 )
   END_RUNG wire#w1
   // the same network as SCL:
   "DB371_M_UNIT_SPARE".M_CODES_SPARE.M623 := ("DB339_EXTENDED_M_SPARE".M_code[623] OR "DB371_M_UNIT_SPARE".M_CODES_SPARE.M623) AND NOT "DB371_M_UNIT_SPARE".M_CODES_SPARE.Ack_M623 AND NOT "DB2120_MPP_ITC_IPC".RESET_FAULTS AND NOT "DB371_M_UNIT_SPARE".M_CODES_SPARE.M_RESET_PULSE;
END_REGION

REGION Network 205: ACKNOWLEDGE M624-FIXTURE 3 GRIPPER RELEASE PRESSURE (READ-IN DISABLE) / ACKNOWLEDGE M112-AXIAL LOCATOR RELAX FIXTURE 1
   RUNG wire#powerrail
      Contact( "DB3710_U2_F3_GRIPPER".PRESSURE_RELEASED )
      Coil( "DB371_M_UNIT_SPARE".M_CODES_SPARE.Ack_M624 )
   END_RUNG
   // the same network as SCL:
   "DB371_M_UNIT_SPARE".M_CODES_SPARE.Ack_M624 := "DB3710_U2_F3_GRIPPER".PRESSURE_RELEASED;
END_REGION

REGION Network 206: M624-FIXTURE 3 GRIPPER RELEASE PRESSURE (READ-IN DISABLE) / M112-AXIAL LOCATOR RELAX FIXTURE 1
   RUNG wire#powerrail
      Contact( "DB339_EXTENDED_M_SPARE".M_code[624] )
      wire#w1
      I_Contact( "DB371_M_UNIT_SPARE".M_CODES_SPARE.Ack_M624 )
      I_Contact( "DB2120_MPP_ITC_IPC".RESET_FAULTS )
      I_Contact( "DB371_M_UNIT_SPARE".M_CODES_SPARE.M_RESET_PULSE )
      Coil( "DB371_M_UNIT_SPARE".M_CODES_SPARE.M624 )
   END_RUNG
   RUNG wire#powerrail
      Contact( "DB371_M_UNIT_SPARE".M_CODES_SPARE.M624 )
   END_RUNG wire#w1
   // the same network as SCL:
   "DB371_M_UNIT_SPARE".M_CODES_SPARE.M624 := ("DB339_EXTENDED_M_SPARE".M_code[624] OR "DB371_M_UNIT_SPARE".M_CODES_SPARE.M624) AND NOT "DB371_M_UNIT_SPARE".M_CODES_SPARE.Ack_M624 AND NOT "DB2120_MPP_ITC_IPC".RESET_FAULTS AND NOT "DB371_M_UNIT_SPARE".M_CODES_SPARE.M_RESET_PULSE;
END_REGION

REGION Network 207: ACKNOWLEDGE M625-FIXTURE 3 GRIPPER LOW PRESSURE (READ-IN DISABLE) / ACKNOWLEDGE M23-SWITCH ON SPINDLE FRAME BLOWING
   RUNG wire#powerrail
      Contact( "DB3710_U2_F3_GRIPPER".CYL.FULL_LOW_PRESSURED )
      Coil( "DB371_M_UNIT_SPARE".M_CODES_SPARE.Ack_M625 )
   END_RUNG
   // the same network as SCL:
   "DB371_M_UNIT_SPARE".M_CODES_SPARE.Ack_M625 := "DB3710_U2_F3_GRIPPER".CYL.FULL_LOW_PRESSURED;
END_REGION

REGION Network 208: M625-FIXTURE 3 GRIPPER LOW PRESSURE (READ-IN DISABLE) / M23-SWITCH ON SPINDLE FRAME BLOWING
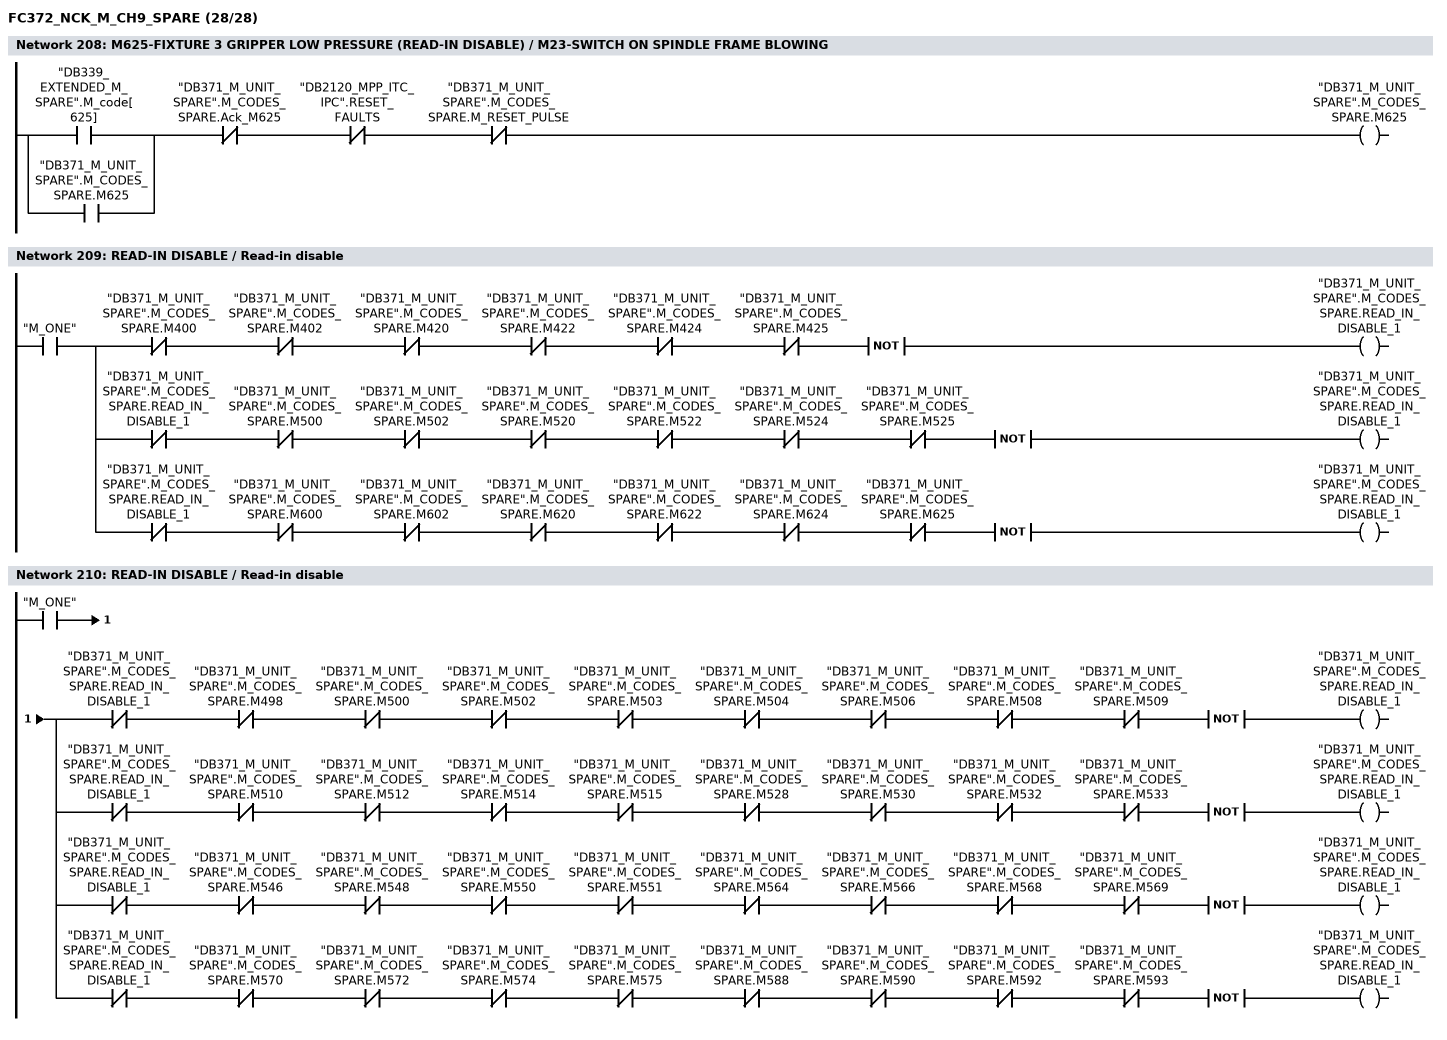
   RUNG wire#powerrail
      Contact( "DB339_EXTENDED_M_SPARE".M_code[625] )
      wire#w1
      I_Contact( "DB371_M_UNIT_SPARE".M_CODES_SPARE.Ack_M625 )
      I_Contact( "DB2120_MPP_ITC_IPC".RESET_FAULTS )
      I_Contact( "DB371_M_UNIT_SPARE".M_CODES_SPARE.M_RESET_PULSE )
      Coil( "DB371_M_UNIT_SPARE".M_CODES_SPARE.M625 )
   END_RUNG
   RUNG wire#powerrail
      Contact( "DB371_M_UNIT_SPARE".M_CODES_SPARE.M625 )
   END_RUNG wire#w1
   // the same network as SCL:
   "DB371_M_UNIT_SPARE".M_CODES_SPARE.M625 := ("DB339_EXTENDED_M_SPARE".M_code[625] OR "DB371_M_UNIT_SPARE".M_CODES_SPARE.M625) AND NOT "DB371_M_UNIT_SPARE".M_CODES_SPARE.Ack_M625 AND NOT "DB2120_MPP_ITC_IPC".RESET_FAULTS AND NOT "DB371_M_UNIT_SPARE".M_CODES_SPARE.M_RESET_PULSE;
END_REGION

REGION Network 209: READ-IN DISABLE / Read-in disable
   RUNG wire#powerrail
      Contact( "M_ONE" )
      wire#w1
      I_Contact( "DB371_M_UNIT_SPARE".M_CODES_SPARE.M400 )
      I_Contact( "DB371_M_UNIT_SPARE".M_CODES_SPARE.M402 )
      I_Contact( "DB371_M_UNIT_SPARE".M_CODES_SPARE.M420 )
      I_Contact( "DB371_M_UNIT_SPARE".M_CODES_SPARE.M422 )
      I_Contact( "DB371_M_UNIT_SPARE".M_CODES_SPARE.M424 )
      I_Contact( "DB371_M_UNIT_SPARE".M_CODES_SPARE.M425 )
      Not()
      Coil( "DB371_M_UNIT_SPARE".M_CODES_SPARE.READ_IN_DISABLE_1 )
   END_RUNG
   RUNG wire#w1
      I_Contact( "DB371_M_UNIT_SPARE".M_CODES_SPARE.READ_IN_DISABLE_1 )
      I_Contact( "DB371_M_UNIT_SPARE".M_CODES_SPARE.M500 )
      I_Contact( "DB371_M_UNIT_SPARE".M_CODES_SPARE.M502 )
      I_Contact( "DB371_M_UNIT_SPARE".M_CODES_SPARE.M520 )
      I_Contact( "DB371_M_UNIT_SPARE".M_CODES_SPARE.M522 )
      I_Contact( "DB371_M_UNIT_SPARE".M_CODES_SPARE.M524 )
      I_Contact( "DB371_M_UNIT_SPARE".M_CODES_SPARE.M525 )
      Not()
      Coil( "DB371_M_UNIT_SPARE".M_CODES_SPARE.READ_IN_DISABLE_1 )
   END_RUNG
   RUNG wire#w1
      I_Contact( "DB371_M_UNIT_SPARE".M_CODES_SPARE.READ_IN_DISABLE_1 )
      I_Contact( "DB371_M_UNIT_SPARE".M_CODES_SPARE.M600 )
      I_Contact( "DB371_M_UNIT_SPARE".M_CODES_SPARE.M602 )
      I_Contact( "DB371_M_UNIT_SPARE".M_CODES_SPARE.M620 )
      I_Contact( "DB371_M_UNIT_SPARE".M_CODES_SPARE.M622 )
      I_Contact( "DB371_M_UNIT_SPARE".M_CODES_SPARE.M624 )
      I_Contact( "DB371_M_UNIT_SPARE".M_CODES_SPARE.M625 )
      Not()
      Coil( "DB371_M_UNIT_SPARE".M_CODES_SPARE.READ_IN_DISABLE_1 )
   END_RUNG
   // the same network as SCL:
   "DB371_M_UNIT_SPARE".M_CODES_SPARE.READ_IN_DISABLE_1 := NOT ("M_ONE" AND NOT "DB371_M_UNIT_SPARE".M_CODES_SPARE.M400 AND NOT "DB371_M_UNIT_SPARE".M_CODES_SPARE.M402 AND NOT "DB371_M_UNIT_SPARE".M_CODES_SPARE.M420 AND NOT "DB371_M_UNIT_SPARE".M_CODES_SPARE.M422 AND NOT "DB371_M_UNIT_SPARE".M_CODES_SPARE.M424 AND NOT "DB371_M_UNIT_SPARE".M_CODES_SPARE.M425);
   "DB371_M_UNIT_SPARE".M_CODES_SPARE.READ_IN_DISABLE_1 := NOT ("M_ONE" AND NOT "DB371_M_UNIT_SPARE".M_CODES_SPARE.READ_IN_DISABLE_1 AND NOT "DB371_M_UNIT_SPARE".M_CODES_SPARE.M500 AND NOT "DB371_M_UNIT_SPARE".M_CODES_SPARE.M502 AND NOT "DB371_M_UNIT_SPARE".M_CODES_SPARE.M520 AND NOT "DB371_M_UNIT_SPARE".M_CODES_SPARE.M522 AND NOT "DB371_M_UNIT_SPARE".M_CODES_SPARE.M524 AND NOT "DB371_M_UNIT_SPARE".M_CODES_SPARE.M525);
   "DB371_M_UNIT_SPARE".M_CODES_SPARE.READ_IN_DISABLE_1 := NOT ("M_ONE" AND NOT "DB371_M_UNIT_SPARE".M_CODES_SPARE.READ_IN_DISABLE_1 AND NOT "DB371_M_UNIT_SPARE".M_CODES_SPARE.M600 AND NOT "DB371_M_UNIT_SPARE".M_CODES_SPARE.M602 AND NOT "DB371_M_UNIT_SPARE".M_CODES_SPARE.M620 AND NOT "DB371_M_UNIT_SPARE".M_CODES_SPARE.M622 AND NOT "DB371_M_UNIT_SPARE".M_CODES_SPARE.M624 AND NOT "DB371_M_UNIT_SPARE".M_CODES_SPARE.M625);
END_REGION

REGION Network 210: READ-IN DISABLE / Read-in disable
   RUNG wire#powerrail
      Contact( "M_ONE" )
      wire#w1
      I_Contact( "DB371_M_UNIT_SPARE".M_CODES_SPARE.READ_IN_DISABLE_1 )
      I_Contact( "DB371_M_UNIT_SPARE".M_CODES_SPARE.M498 )
      I_Contact( "DB371_M_UNIT_SPARE".M_CODES_SPARE.M500 )
      I_Contact( "DB371_M_UNIT_SPARE".M_CODES_SPARE.M502 )
      I_Contact( "DB371_M_UNIT_SPARE".M_CODES_SPARE.M503 )
      I_Contact( "DB371_M_UNIT_SPARE".M_CODES_SPARE.M504 )
      I_Contact( "DB371_M_UNIT_SPARE".M_CODES_SPARE.M506 )
      I_Contact( "DB371_M_UNIT_SPARE".M_CODES_SPARE.M508 )
      I_Contact( "DB371_M_UNIT_SPARE".M_CODES_SPARE.M509 )
      Not()
      Coil( "DB371_M_UNIT_SPARE".M_CODES_SPARE.READ_IN_DISABLE_1 )
   END_RUNG
   RUNG wire#w1
      I_Contact( "DB371_M_UNIT_SPARE".M_CODES_SPARE.READ_IN_DISABLE_1 )
      I_Contact( "DB371_M_UNIT_SPARE".M_CODES_SPARE.M510 )
      I_Contact( "DB371_M_UNIT_SPARE".M_CODES_SPARE.M512 )
      I_Contact( "DB371_M_UNIT_SPARE".M_CODES_SPARE.M514 )
      I_Contact( "DB371_M_UNIT_SPARE".M_CODES_SPARE.M515 )
      I_Contact( "DB371_M_UNIT_SPARE".M_CODES_SPARE.M528 )
      I_Contact( "DB371_M_UNIT_SPARE".M_CODES_SPARE.M530 )
      I_Contact( "DB371_M_UNIT_SPARE".M_CODES_SPARE.M532 )
      I_Contact( "DB371_M_UNIT_SPARE".M_CODES_SPARE.M533 )
      Not()
      Coil( "DB371_M_UNIT_SPARE".M_CODES_SPARE.READ_IN_DISABLE_1 )
   END_RUNG
   RUNG wire#w1
      I_Contact( "DB371_M_UNIT_SPARE".M_CODES_SPARE.READ_IN_DISABLE_1 )
      I_Contact( "DB371_M_UNIT_SPARE".M_CODES_SPARE.M546 )
      I_Contact( "DB371_M_UNIT_SPARE".M_CODES_SPARE.M548 )
      I_Contact( "DB371_M_UNIT_SPARE".M_CODES_SPARE.M550 )
      I_Contact( "DB371_M_UNIT_SPARE".M_CODES_SPARE.M551 )
      I_Contact( "DB371_M_UNIT_SPARE".M_CODES_SPARE.M564 )
      I_Contact( "DB371_M_UNIT_SPARE".M_CODES_SPARE.M566 )
      I_Contact( "DB371_M_UNIT_SPARE".M_CODES_SPARE.M568 )
      I_Contact( "DB371_M_UNIT_SPARE".M_CODES_SPARE.M569 )
      Not()
      Coil( "DB371_M_UNIT_SPARE".M_CODES_SPARE.READ_IN_DISABLE_1 )
   END_RUNG
   RUNG wire#w1
      I_Contact( "DB371_M_UNIT_SPARE".M_CODES_SPARE.READ_IN_DISABLE_1 )
      I_Contact( "DB371_M_UNIT_SPARE".M_CODES_SPARE.M570 )
      I_Contact( "DB371_M_UNIT_SPARE".M_CODES_SPARE.M572 )
      I_Contact( "DB371_M_UNIT_SPARE".M_CODES_SPARE.M574 )
      I_Contact( "DB371_M_UNIT_SPARE".M_CODES_SPARE.M575 )
      I_Contact( "DB371_M_UNIT_SPARE".M_CODES_SPARE.M588 )
      I_Contact( "DB371_M_UNIT_SPARE".M_CODES_SPARE.M590 )
      I_Contact( "DB371_M_UNIT_SPARE".M_CODES_SPARE.M592 )
      I_Contact( "DB371_M_UNIT_SPARE".M_CODES_SPARE.M593 )
      Not()
      Coil( "DB371_M_UNIT_SPARE".M_CODES_SPARE.READ_IN_DISABLE_1 )
   END_RUNG
   // the same network as SCL:
   "DB371_M_UNIT_SPARE".M_CODES_SPARE.READ_IN_DISABLE_1 := NOT ("M_ONE" AND NOT "DB371_M_UNIT_SPARE".M_CODES_SPARE.READ_IN_DISABLE_1 AND NOT "DB371_M_UNIT_SPARE".M_CODES_SPARE.M498 AND NOT "DB371_M_UNIT_SPARE".M_CODES_SPARE.M500 AND NOT "DB371_M_UNIT_SPARE".M_CODES_SPARE.M502 AND NOT "DB371_M_UNIT_SPARE".M_CODES_SPARE.M503 AND NOT "DB371_M_UNIT_SPARE".M_CODES_SPARE.M504 AND NOT "DB371_M_UNIT_SPARE".M_CODES_SPARE.M506 AND NOT "DB371_M_UNIT_SPARE".M_CODES_SPARE.M508 AND NOT "DB371_M_UNIT_SPARE".M_CODES_SPARE.M509);
   "DB371_M_UNIT_SPARE".M_CODES_SPARE.READ_IN_DISABLE_1 := NOT ("M_ONE" AND NOT "DB371_M_UNIT_SPARE".M_CODES_SPARE.READ_IN_DISABLE_1 AND NOT "DB371_M_UNIT_SPARE".M_CODES_SPARE.M510 AND NOT "DB371_M_UNIT_SPARE".M_CODES_SPARE.M512 AND NOT "DB371_M_UNIT_SPARE".M_CODES_SPARE.M514 AND NOT "DB371_M_UNIT_SPARE".M_CODES_SPARE.M515 AND NOT "DB371_M_UNIT_SPARE".M_CODES_SPARE.M528 AND NOT "DB371_M_UNIT_SPARE".M_CODES_SPARE.M530 AND NOT "DB371_M_UNIT_SPARE".M_CODES_SPARE.M532 AND NOT "DB371_M_UNIT_SPARE".M_CODES_SPARE.M533);
   "DB371_M_UNIT_SPARE".M_CODES_SPARE.READ_IN_DISABLE_1 := NOT ("M_ONE" AND NOT "DB371_M_UNIT_SPARE".M_CODES_SPARE.READ_IN_DISABLE_1 AND NOT "DB371_M_UNIT_SPARE".M_CODES_SPARE.M546 AND NOT "DB371_M_UNIT_SPARE".M_CODES_SPARE.M548 AND NOT "DB371_M_UNIT_SPARE".M_CODES_SPARE.M550 AND NOT "DB371_M_UNIT_SPARE".M_CODES_SPARE.M551 AND NOT "DB371_M_UNIT_SPARE".M_CODES_SPARE.M564 AND NOT "DB371_M_UNIT_SPARE".M_CODES_SPARE.M566 AND NOT "DB371_M_UNIT_SPARE".M_CODES_SPARE.M568 AND NOT "DB371_M_UNIT_SPARE".M_CODES_SPARE.M569);
   "DB371_M_UNIT_SPARE".M_CODES_SPARE.READ_IN_DISABLE_1 := NOT ("M_ONE" AND NOT "DB371_M_UNIT_SPARE".M_CODES_SPARE.READ_IN_DISABLE_1 AND NOT "DB371_M_UNIT_SPARE".M_CODES_SPARE.M570 AND NOT "DB371_M_UNIT_SPARE".M_CODES_SPARE.M572 AND NOT "DB371_M_UNIT_SPARE".M_CODES_SPARE.M574 AND NOT "DB371_M_UNIT_SPARE".M_CODES_SPARE.M575 AND NOT "DB371_M_UNIT_SPARE".M_CODES_SPARE.M588 AND NOT "DB371_M_UNIT_SPARE".M_CODES_SPARE.M590 AND NOT "DB371_M_UNIT_SPARE".M_CODES_SPARE.M592 AND NOT "DB371_M_UNIT_SPARE".M_CODES_SPARE.M593);
END_REGION
END_FUNCTION
